// SIMATIC STEP 7 (V5.x) project S_M_Cizallado
// CPU: CPU312(1)
// station: P_ADR_BUS
// station: Hardware
// station: Equipo SIMATIC 300
// program: Programa S7(1)

SYMBOL_TABLE
"CONTADOR"	C 1	COUNTER
"CIZALLADO"	FB 2	FB 2	// Funcion que se encaga del cizallado de planchas
"MULT_CIZA"	FB 4	FB 4
"CORTAR"	FC 1	FC 1	// Funcion de cortar las planchas
"S_CACEROLA"	I 124.0	BOOL
"S_SARTEN"	I 124.1	BOOL
"S_PAELLERA"	I 124.2	BOOL
"S_WOK"	I 124.3	BOOL
"BIT_DE_TRABAJO"	I 124.4	BOOL
"SENSORARRIBA"	I 124.6	BOOL
"SENSORABAJO"	I 124.7	BOOL
"EXPULSADA"	I 125.0	BOOL
"START"	I 125.1	BOOL
"LOAD_CONT"	I 125.2	BOOL
"SARTEN"	I 125.3	BOOL
"CACEROLA"	I 125.4	BOOL
"WOK"	I 125.5	BOOL
"PAELLERA"	I 125.6	BOOL
"Cycle Execution"	OB 1	OB 1
"PLANCHAS"	PIW 651	INT
"EXPULSARPLANCHA"	Q 100.1	BOOL
"BAJARCUCHILLA"	Q 100.2	BOOL
"BIT_OK"	Q 100.3	BOOL
"STBY"	Q 100.4	BOOL
END_SYMBOL_TABLE

FUNCTION_BLOCK "CIZALLADO"	// FB 2
TITLE = CIZALLADO
VERSION : 0.1
VAR_INPUT
  bit_de_trabajo : BOOL ;
  SENSOR : BOOL ;
  SENSORABAJO : BOOL ;
  SENSORARRIBA : BOOL ;
  EXPULSADA : BOOL ;
  CONTADOR : COUNTER ;
  START : BOOL ;
END_VAR
VAR_OUTPUT
  BAJARCUCHILLA : BOOL ;
  EXPULSARPLANCHA : BOOL ;
  STBY : BOOL ;
  BIT_OK : BOOL ;
END_VAR
VAR
  X41 : BOOL ;
  M3 : BOOL ;
  X43 : BOOL ;
  FP_BDT : BOOL ;
  FP_START : BOOL ;
  INICORTAR : BOOL ;
  S2 : BOOL ;
  BDT_CORTAR : BOOL ;
  OK_CORTAR : BOOL ;
  STBY_CORTAR : BOOL ;
  CORTADO : BOOL ;
END_VAR
BEGIN
NETWORK
TITLE = Arranque
      A     #bit_de_trabajo;
      FP    #FP_BDT;
      =     #BDT_CORTAR;
      S     #X41;
      R     #M3;
      R     #X43;
      R     #INICORTAR;
      R     #CORTADO;
      R     #BIT_OK;
      R     #S2;
NETWORK
TITLE = De x41 a M3
      A     #X41;
      A     #SENSOR;
      A     #STBY_CORTAR;
      A     #START;
      FP    #FP_START;
      R     #X41;
      S     #M3;
NETWORK
TITLE = De M3 a x43
      A     #M3;
      A     #CORTADO;
      R     #M3;
      S     #X43;
NETWORK
TITLE = de x43 a x41
      A     #X43;
      T     LD 0;
      TAK;
      T     LD 4;
      L     #CONTADOR;
      T     LW 8;
      L     LD 4;
      L     LD 0;
      AN    C [LW 8];
      R     #X43;
      S     #S2;
NETWORK
TITLE = de x43 a X41
      A     #X43;
      T     LD 0;
      TAK;
      T     LD 4;
      L     #CONTADOR;
      T     LW 8;
      L     LD 4;
      L     LD 0;
      A     C [LW 8];
      R     #X43;
      S     #X41;
NETWORK
TITLE = De M3 a x43 con call M3
      CALL  "CORTAR" (
           bit_de_trabajo           := #BDT_CORTAR,
           SENSORABAJO              := #SENSORABAJO,
           SENSORARRIBA             := #SENSORARRIBA,
           EXPULSADA                := #EXPULSADA,
           START                    := #INICORTAR,
           OK                       := #OK_CORTAR,
           BAJARCUCHILLA            := #BAJARCUCHILLA,
           EXPULSARPLANCHA          := #EXPULSARPLANCHA,
           bit_ok                   := #CORTADO,
           STBY                     := #STBY_CORTAR);
NETWORK
TITLE =
      A     #M3;
      A     #CORTADO;
      R     #M3;
      S     #X43;
NETWORK
TITLE =
      A     #M3;
      =     #INICORTAR;
NETWORK
TITLE = Cuenta el numero de planchas cortadas
      A     #X43;
      =     #OK_CORTAR;
      T     LD 0;
      TAK;
      T     LD 4;
      L     #CONTADOR;
      T     LW 8;
      L     LD 4;
      L     LD 0;
      CD    C [LW 8];
NETWORK
TITLE =
      A     #X41;
      =     #STBY;
NETWORK
TITLE =
      A     #S2;
      =     #BIT_OK;
END_FUNCTION_BLOCK

FUNCTION_BLOCK "MULT_CIZA"	// FB 4
VERSION : 0.1
VAR_INPUT
  S_CACEROLA : BOOL ;
  S_WOK : BOOL ;
  S_SARTEN : BOOL ;
  S_PAELLERA : BOOL ;
  BIT_DE_TRABAJO : BOOL ;
  SENSORARRIBA : BOOL ;
  SENSORABAJO : BOOL ;
  EXPULSADA : BOOL ;
  CONTADOR : COUNTER ;
  SARTEN : BOOL ;
  CACEROLA : BOOL ;
  WOK : BOOL ;
  PAELLERA : BOOL ;
  START : BOOL ;
END_VAR
VAR_OUTPUT
  EXPULSARPLANCHA : BOOL ;
  BAJARCUCHILLA : BOOL ;
  BIT_OK : BOOL ;
  STBY : BOOL ;
END_VAR
VAR
  BDT : BOOL ;
  START_SAR : BOOL ;
  START_CAC : BOOL ;
  START_WOK : BOOL ;
  START_PAELL : BOOL ;
  X1 : BOOL ;
  X2 : BOOL ;
  X3 : BOOL ;
  X4 : BOOL ;
  X5 : BOOL ;
  FP_START : BOOL ;
  F_START : BOOL ;
  STBY_SAR : BOOL ;
  STBY_CAC : BOOL ;
  STBY_WOK : BOOL ;
  STBY_PAELL : BOOL ;
  OK : BOOL ;
  FP_BDT : BOOL ;
  CAC_CIZA : FB 2;
  SART_CIZA : FB 2;
  WOK_CIZA : FB 2;
  PAELL_CIZA : FB 2;
  X6 : BOOL ;
  FP_OK : BOOL ;
END_VAR
BEGIN
NETWORK
TITLE =
      A     #BIT_DE_TRABAJO;
      FP    #FP_BDT;
      S     #X1;
      R     #X2;
      R     #X3;
      R     #X4;
      R     #X5;
      R     #X6;
NETWORK
TITLE =
      A     #START;
      FP    #FP_START;
      =     #F_START;
NETWORK
TITLE =
      A     #F_START;
      A     #SARTEN;
      A     #X1;
      R     #X1;
      S     #X2;
NETWORK
TITLE =
      A     #F_START;
      A     #CACEROLA;
      A     #X1;
      R     #X1;
      S     #X3;
NETWORK
TITLE =
      A     #F_START;
      A     #WOK;
      A     #X1;
      R     #X1;
      S     #X4;
NETWORK
TITLE =
      A     #F_START;
      A     #PAELLERA;
      A     #X1;
      R     #X1;
      S     #X5;
NETWORK
TITLE =
      A     #OK;
      FP    #FP_OK;
      A(;
      O     #X2;
      O     #X3;
      O     #X4;
      O     #X5;
      );
      R     #X2;
      R     #X3;
      R     #X4;
      R     #X5;
      S     #X6;
NETWORK
TITLE =
      A     #X2;
      JCN   _001;
      S     #BDT;
      BLD   14;
      =     L 6.0;
      L     DINO;
      T     LW 4;
      CDB;
      OPN   DI [LW 4];
      TAR2  LD 0;
      A     DBX [AR2,P#8.0];
      =     #SART_CIZA.bit_de_trabajo;
      A     DBX [AR2,P#0.2];
      =     #SART_CIZA.SENSOR;
      A     DBX [AR2,P#0.6];
      =     #SART_CIZA.SENSORABAJO;
      A     DBX [AR2,P#0.5];
      =     #SART_CIZA.SENSORARRIBA;
      A     DBX [AR2,P#0.7];
      =     #SART_CIZA.EXPULSADA;
      L     DBW [AR2,P#2.0];
      T     #SART_CIZA.CONTADOR;
      A     DBX [AR2,P#4.4];
      =     #SART_CIZA.START;
      +AR2  P#22.0;
      UC    "CIZALLADO";
      LAR2  LD 0;
      A     #SART_CIZA.BAJARCUCHILLA;
      =     DBX [AR2,P#6.1];
      A     #SART_CIZA.EXPULSARPLANCHA;
      =     DBX [AR2,P#6.0];
      A     #SART_CIZA.STBY;
      =     DBX [AR2,P#6.3];
      A     #SART_CIZA.BIT_OK;
      =     DBX [AR2,P#10.0];
      CDB;
      BLD   15;
_001: NOP   0;
NETWORK
TITLE =
      A     #X3;
      JCN   _002;
      S     #BDT;
      BLD   14;
      =     L 6.0;
      L     DINO;
      T     LW 4;
      CDB;
      OPN   DI [LW 4];
      TAR2  LD 0;
      A     DBX [AR2,P#8.0];
      =     #CAC_CIZA.bit_de_trabajo;
      A     DBX [AR2,P#0.0];
      =     #CAC_CIZA.SENSOR;
      A     DBX [AR2,P#0.6];
      =     #CAC_CIZA.SENSORABAJO;
      A     DBX [AR2,P#0.5];
      =     #CAC_CIZA.SENSORARRIBA;
      A     DBX [AR2,P#0.7];
      =     #CAC_CIZA.EXPULSADA;
      L     DBW [AR2,P#2.0];
      T     #CAC_CIZA.CONTADOR;
      A     DBX [AR2,P#4.4];
      =     #CAC_CIZA.START;
      +AR2  P#12.0;
      UC    "CIZALLADO";
      LAR2  LD 0;
      A     #CAC_CIZA.BAJARCUCHILLA;
      =     DBX [AR2,P#6.1];
      A     #CAC_CIZA.EXPULSARPLANCHA;
      =     DBX [AR2,P#6.0];
      A     #CAC_CIZA.STBY;
      =     DBX [AR2,P#6.3];
      A     #CAC_CIZA.BIT_OK;
      =     DBX [AR2,P#10.0];
      CDB;
      BLD   15;
_002: NOP   0;
NETWORK
TITLE =
      A     #X4;
      JCN   _003;
      S     #BDT;
      BLD   14;
      =     L 6.0;
      L     DINO;
      T     LW 4;
      CDB;
      OPN   DI [LW 4];
      TAR2  LD 0;
      A     DBX [AR2,P#8.0];
      =     #WOK_CIZA.bit_de_trabajo;
      A     DBX [AR2,P#0.1];
      =     #WOK_CIZA.SENSOR;
      A     DBX [AR2,P#0.6];
      =     #WOK_CIZA.SENSORABAJO;
      A     DBX [AR2,P#0.5];
      =     #WOK_CIZA.SENSORARRIBA;
      A     DBX [AR2,P#0.7];
      =     #WOK_CIZA.EXPULSADA;
      L     DBW [AR2,P#2.0];
      T     #WOK_CIZA.CONTADOR;
      A     DBX [AR2,P#4.4];
      =     #WOK_CIZA.START;
      +AR2  P#32.0;
      UC    "CIZALLADO";
      LAR2  LD 0;
      A     #WOK_CIZA.BAJARCUCHILLA;
      =     DBX [AR2,P#6.1];
      A     #WOK_CIZA.EXPULSARPLANCHA;
      =     DBX [AR2,P#6.0];
      A     #WOK_CIZA.STBY;
      =     DBX [AR2,P#6.3];
      A     #WOK_CIZA.BIT_OK;
      =     DBX [AR2,P#10.0];
      CDB;
      BLD   15;
_003: NOP   0;
NETWORK
TITLE =
      A     #X5;
      JCN   _004;
      S     #BDT;
      BLD   14;
      =     L 6.0;
      L     DINO;
      T     LW 4;
      CDB;
      OPN   DI [LW 4];
      TAR2  LD 0;
      A     DBX [AR2,P#8.0];
      =     #PAELL_CIZA.bit_de_trabajo;
      A     DBX [AR2,P#0.3];
      =     #PAELL_CIZA.SENSOR;
      A     DBX [AR2,P#0.6];
      =     #PAELL_CIZA.SENSORABAJO;
      A     DBX [AR2,P#0.5];
      =     #PAELL_CIZA.SENSORARRIBA;
      A     DBX [AR2,P#0.7];
      =     #PAELL_CIZA.EXPULSADA;
      L     DBW [AR2,P#2.0];
      T     #PAELL_CIZA.CONTADOR;
      A     DBX [AR2,P#4.4];
      =     #PAELL_CIZA.START;
      +AR2  P#42.0;
      UC    "CIZALLADO";
      LAR2  LD 0;
      A     #PAELL_CIZA.BAJARCUCHILLA;
      =     DBX [AR2,P#6.1];
      A     #PAELL_CIZA.EXPULSARPLANCHA;
      =     DBX [AR2,P#6.0];
      A     #PAELL_CIZA.STBY;
      =     DBX [AR2,P#6.3];
      A     #PAELL_CIZA.BIT_OK;
      =     DBX [AR2,P#10.0];
      CDB;
      BLD   15;
_004: NOP   0;
NETWORK
TITLE =
      A     #X2;
      =     #START_SAR;
NETWORK
TITLE =
      A     #X3;
      =     #START_CAC;
NETWORK
TITLE =
      A     #X4;
      =     #START_WOK;
NETWORK
TITLE =
      A     #X5;
      =     #START_PAELL;
NETWORK
TITLE =
      A     #X1;
      =     #STBY;
NETWORK
TITLE =
      A     #X6;
      =     #BIT_OK;
      R     #BDT;
      R     #OK;
END_FUNCTION_BLOCK

FUNCTION "CORTAR" : VOID	// FC 1
TITLE = CORTAR
VERSION : 0.1
VAR_INPUT
  bit_de_trabajo : BOOL ;
  SENSORABAJO : BOOL ;
  SENSORARRIBA : BOOL ;
  EXPULSADA : BOOL ;
  START : BOOL ;
  OK : BOOL ;
END_VAR
VAR_OUTPUT
  BAJARCUCHILLA : BOOL ;
  EXPULSARPLANCHA : BOOL ;
  bit_ok : BOOL ;
  STBY : BOOL ;
END_VAR
VAR_TEMP
  x51 : BOOL ;
  x52 : BOOL ;
  x53 : BOOL ;
  s3 : BOOL ;
  FP_BDT : BOOL ;
  X50 : BOOL ;
  FP_START : BOOL ;
END_VAR
BEGIN
NETWORK
TITLE = Arranque
      A     #bit_de_trabajo;
      FP    #FP_BDT;
      S     #X50;
      R     #x51;
      R     #x52;
      R     #x53;
      R     #s3;
NETWORK
TITLE = de x51 a x52
      A     #x51;
      A     #SENSORABAJO;
      R     #x51;
      S     #x52;
NETWORK
TITLE = de x52 a x53
      A     #x52;
      A     #SENSORARRIBA;
      R     #x52;
      S     #x53;
NETWORK
TITLE = de x53 a s3
      A     #x53;
      A     #EXPULSADA;
      R     #x53;
      S     #s3;
NETWORK
TITLE = Accion x51
      A     #x51;
      =     #BAJARCUCHILLA;
NETWORK
TITLE = Accion x53
      A     #x53;
      =     #EXPULSARPLANCHA;
NETWORK
TITLE = Accion final
      A     #s3;
      =     #bit_ok;
NETWORK
TITLE =
      A     #s3;
      A     #OK;
      R     #s3;
      S     #X50;
NETWORK
TITLE =
      A     #X50;
      A     #START;
      FP    #FP_START;
      R     #X50;
      S     #x51;
NETWORK
TITLE =
      A     #X50;
      =     #STBY;
END_FUNCTION

DATA_BLOCK DB 1
VERSION : 0.0
"MULT_CIZA"
BEGIN
END_DATA_BLOCK

ORGANIZATION_BLOCK "Cycle Execution"	// OB 1
TITLE = "Main Program Sweep (Cycle)"
VERSION : 0.1
VAR_TEMP
  OB1_EV_CLASS : BYTE ;	//Bits 0-3 = 1 (Coming event), Bits 4-7 = 1 (Event class 1)
  OB1_SCAN_1 : BYTE ;	//1 (Cold restart scan 1 of OB 1), 3 (Scan 2-n of OB 1)
  OB1_PRIORITY : BYTE ;	//Priority of OB Execution
  OB1_OB_NUMBR : BYTE ;	//1 (Organization block 1, OB1)
  OB1_RESERVED_1 : BYTE ;	//Reserved for system
  OB1_RESERVED_2 : BYTE ;	//Reserved for system
  OB1_PREV_CYCLE : INT ;	//Cycle time of previous OB1 scan (milliseconds)
  OB1_MIN_CYCLE : INT ;	//Minimum cycle time of OB1 (milliseconds)
  OB1_MAX_CYCLE : INT ;	//Maximum cycle time of OB1 (milliseconds)
  OB1_DATE_TIME : DATE_AND_TIME ;	//Date and time OB1 started
END_VAR
BEGIN
NETWORK
TITLE =
      CALL  "MULT_CIZA" , DB 1 (
           S_CACEROLA               := "S_CACEROLA",
           S_WOK                    := "S_WOK",
           S_SARTEN                 := "S_SARTEN",
           S_PAELLERA               := "S_PAELLERA",
           BIT_DE_TRABAJO           := "BIT_DE_TRABAJO",
           SENSORARRIBA             := "SENSORARRIBA",
           SENSORABAJO              := "SENSORABAJO",
           EXPULSADA                := "EXPULSADA",
           CONTADOR                 := "CONTADOR",
           SARTEN                   := "SARTEN",
           CACEROLA                 := "CACEROLA",
           WOK                      := "WOK",
           PAELLERA                 := "PAELLERA",
           START                    := "START",
           EXPULSARPLANCHA          := "EXPULSARPLANCHA",
           BAJARCUCHILLA            := "BAJARCUCHILLA",
           BIT_OK                   := "BIT_OK",
           STBY                     := "STBY");
NETWORK
TITLE =
      A     "LOAD_CONT";
      JCN   _010;
      L     "PLANCHAS";
      S     "CONTADOR";
_010: NOP   0;
END_ORGANIZATION_BLOCK
